FUNCTION_BLOCK FB_BLINK
VAR_INPUT
	ENABLE:		BOOL;
	ON_TIME:	TIME := T#500MS;
	OFF_TIME:	TIME := T#500MS;
END_VAR
VAR_OUTPUT
	Q:		BOOL;
END_VAR
VAR
    IMPULS   :TOF;
    PAUSE    :TOF;
END_VAR

IMPULS(IN:= NOT PAUSE.Q AND NOT IMPULS.Q, PT:= ON_TIME);
PAUSE(IN:= NOT PAUSE.Q AND NOT IMPULS.Q, PT:= OFF_TIME);
Q := IMPULS.Q AND ENABLE;

END_FUNCTION_BLOCK

(* stored: Version 1.1.0.1, ProductVersion 3.1.4024.0
   POU FB_BLINK: Id {56aa9b26-e1df-4289-b787-9e9311227a5a}, SpecialFunc None *)
